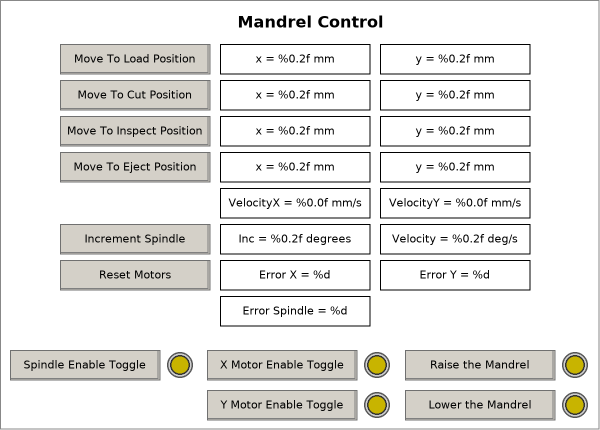
VISUALIZATION Manual_Mandrel  // 600x430
    Button (60,44 150x30), "Move To Load Position", input disabled if: MAIN.fbSlitter.bBusy
        OnMouseClick: execute { MAIN.fbSlitter.Manual.bMoveToLoadPosition := TRUE; }
    Button (60,80 150x30), "Move To Cut Position", input disabled if: MAIN.fbSlitter.bBusy
        OnMouseClick: execute { MAIN.fbSlitter.Manual.bMoveToCutPosition := TRUE; }
    Button (60,116 150x30), "Move To Inspect Position", input disabled if: MAIN.fbSlitter.bBusy
        OnMouseClick: execute { MAIN.fbSlitter.Manual.bMoveToInspectPosition := TRUE; }
    Button (60,152 150x30), "Move To Eject Position", input disabled if: MAIN.fbSlitter.bBusy
        OnMouseClick: execute { MAIN.fbSlitter.Manual.bMoveToEjectPosition := TRUE; }
    Button (405,350 150x30), "Raise the Mandrel", input disabled if: MAIN.fbSlitter.bBusy
        OnMouseClick: execute { MAIN.fbSlitter.Manual.bRaiseMandrel := TRUE; }
    Button (405,390 150x30), "Lower the Mandrel", input disabled if: MAIN.fbSlitter.bBusy
        OnMouseClick: execute { MAIN.fbSlitter.Manual.bLowerMandrel := TRUE; }
    Rectangle (220,44 150x30), "x = %0.2f mm", text variable: MAIN.fbSlitter.Mandrel._hmiParameters.loadPositionX
        OnMouseClick: write MAIN.fbSlitter.Mandrel._hmiParameters.loadPositionX via Default, title 'Load Position X'
    Rectangle (380,44 150x30), "y = %0.2f mm", text variable: MAIN.fbSlitter.Mandrel._hmiParameters.loadPositionY
        OnMouseClick: write MAIN.fbSlitter.Mandrel._hmiParameters.loadPositionY via Default, title 'Load Position Y'
    Rectangle (220,80 150x30), "x = %0.2f mm", text variable: MAIN.TubeHmi.CutPositionX
        OnMouseClick: write MAIN.TubeHmi.CutPositionX via Default, title 'Cut Position X'
    Rectangle (380,80 150x30), "y = %0.2f mm", text variable: MAIN.TubeHmi.CutPositionY
        OnMouseClick: write MAIN.TubeHmi.CutPositionY via Default, title 'Cut Position Y'
    Rectangle (220,116 150x30), "x = %0.2f mm", text variable: MAIN.TubeHmi.InspectPositionX
        OnMouseClick: write MAIN.TubeHmi.InspectPositionX via Default, title 'Inspect Position X'
    Rectangle (380,116 150x30), "y = %0.2f mm", text variable: MAIN.TubeHmi.InspectPositionY
        OnMouseClick: write MAIN.TubeHmi.InspectPositionY via Default, title 'Inspect Position Y'
    Rectangle (220,152 150x30), "x = %0.2f mm", text variable: MAIN.TubeHmi.EjectPositionX
        OnMouseClick: write MAIN.TubeHmi.EjectPositionX via Default, title 'Eject Position X'
    Rectangle (380,152 150x30), "y = %0.2f mm", text variable: MAIN.TubeHmi.EjectPositionY
        OnMouseClick: write MAIN.TubeHmi.EjectPositionY via Default, title 'Eject Position Y'
    Lamp1 (560,350 30x30), variable: MAIN.fbSlitter.Mandrel.doStripperExtend AND NOT MAIN.fbSlitter.Mandrel.doStripperRetract, style: Lamp-Lamp1-Yellow
    Lamp1 (560,390 30x30), variable: NOT MAIN.fbSlitter.Mandrel.doStripperExtend AND MAIN.fbSlitter.Mandrel.doStripperRetract, style: Lamp-Lamp1-Yellow
    Rectangle (220,188 150x30), "VelocityX = %0.0f mm/s", text variable: MAIN.fbSlitter.Mandrel._hmiParameters.velocityX
        OnMouseClick: write MAIN.fbSlitter.Mandrel._hmiParameters.velocityX via Default, title 'Velocity X'
    Rectangle (380,188 150x30), "VelocityY = %0.0f mm/s", text variable: MAIN.fbSlitter.Mandrel._hmiParameters.velocityY
        OnMouseClick: write MAIN.fbSlitter.Mandrel._hmiParameters.velocityY via Default, title 'Velocity Y'
    Rectangle (220,260 150x30), "Error X = %d", text variable: MAIN.fbSlitter.Mandrel.Xaxis.NcToPlc.ErrorCode
    Rectangle (380,260 150x30), "Error Y = %d", text variable: MAIN.fbSlitter.Mandrel.Yaxis.NcToPlc.ErrorCode
    Button (60,260 150x30), "Reset Motors"
        OnMouseClick: execute { MAIN.fbSlitter.Manual.bMandrelReset := TRUE; }
    Button (207,350 150x30), "X Motor Enable Toggle", input disabled if: MAIN.fbSlitter.bBusy
        OnMouseClick: execute { MAIN.fbSlitter.Manual.bMandrelXEnableToggle := TRUE; }
    Button (207,390 150x30), "Y Motor Enable Toggle", input disabled if: MAIN.fbSlitter.bBusy
        OnMouseClick: execute { MAIN.fbSlitter.Manual.bMandrelYEnableToggle := TRUE; }
    Button (10,350 150x30), "Spindle Enable Toggle"
        OnMouseClick: execute { MAIN.fbSlitter.Manual.bMandrelSpindleToggle := TRUE; }
    Lamp1 (362,350 30x30), variable: MAIN.fbSlitter.Mandrel.Xaxis.NcToPlc.StateDWord.0 = 1, style: Lamp-Lamp1-Yellow
    Lamp1 (165,350 30x30), variable: MAIN.fbSlitter.Mandrel.Spindle.NcToPlc.StateDWord.0 = 1, style: Lamp-Lamp1-Yellow
    Lamp1 (362,390 30x30), variable: MAIN.fbSlitter.Mandrel.Yaxis.NcToPlc.StateDWord.0 = 1, style: Lamp-Lamp1-Yellow
    Label (133,7 355x30), "Mandrel Control"
    Rectangle (220,296 150x30), "Error Spindle = %d", text variable: MAIN.fbSlitter.Mandrel.Spindle.NcToPlc.ErrorCode
    Button (60,224 150x30), "Increment Spindle", input disabled if: MAIN.fbSlitter.bBusy
        OnMouseClick: execute { MAIN.fbSlitter.Manual.bMandrelSpindleRotate := TRUE; }
    Rectangle (220,224 150x30), "Inc = %0.2f degrees", text variable: MAIN.fbSlitter.Mandrel._SpindleIncrement
        OnMouseClick: write MAIN.fbSlitter.Mandrel._SpindleIncrement via Default, title 'Spingle Increment'
    Rectangle (380,224 150x30), "Velocity = %0.2f deg/s", text variable: MAIN.fbSlitter.Mandrel._hmiParameters.spindleVelocity
        OnMouseClick: write MAIN.fbSlitter.Mandrel._hmiParameters.spindleVelocity via Default, title 'Spindle Velocity'
END_VISUALIZATION

(* stored: Version 1.1.0.1, ProductVersion 3.1.4024.9
   Visu Manual_Mandrel: Id {41509b5c-e9aa-4eca-bc58-21aad11008db} *)
